// TIA Portal V19 export
FUNCTION "Prod_O_ACT_Pop_&_O_TODO_Push" : DInt   // FC63, LAD
TITLE = POP ORDINE IN LAVORO (ACT) SU ARRAY ORDINI DA FARE (TODO)
// stored: SetENOAutomatically false
   VAR_TEMP
      RETVAL : DInt;
   END_VAR
BEGIN

REGION Network 1 (SCL): SPOSTA ACT SU TODO

   //@@@@@@@@@@@@@@@@@@@@@@@@@@@@@@@@@@@@@@@@@@@@@@@@@@@@@@@@@@@@@@@@@@@@@@@@@@@@@@@@@@@
   //
   // PUSH
   // 
   //@@@@@@@@@@@@@@@@@@@@@@@@@@@@@@@@@@@@@@@@@@@@@@@@@@@@@@@@@@@@@@@@@@@@@@@@@@@@@@@@@@@


   #RETVAL :="PROD_item_Push_to_Top"(item := "Production".O_ACT , Evaluate_FULL := true, Buffer := "Production".O_TODO);


   IF #RETVAL < 0 THEN

       #"Prod_O_ACT_Pop_&_O_TODO_Push" := #RETVAL;

   END_IF;



   //@@@@@@@@@@@@@@@@@@@@@@@@@@@@@@@@@@@@@@@@@@@@@@@@@@@@@@@@@@@@@@@@@@@@@@@@@@@@@@@@@@@
   //
   // POP
   // 
   //@@@@@@@@@@@@@@@@@@@@@@@@@@@@@@@@@@@@@@@@@@@@@@@@@@@@@@@@@@@@@@@@@@@@@@@@@@@@@@@@@@@


   #RETVAL := "Prod_O_ACT_Pop"();


   // Uscita per errore OP
   // 
   IF #RETVAL < 0 THEN

       #"Prod_O_ACT_Pop_&_O_TODO_Push" := #RETVAL;

   END_IF;



   //@@@@@@@@@@@@@@@@@@@@@@@@@@@@@@@@@@@@@@@@@@@@@@@@@@@@@@@@@@@@@@@@@@@@@@@@@@@@@@@@@@@
   //
   // OK
   // 
   //@@@@@@@@@@@@@@@@@@@@@@@@@@@@@@@@@@@@@@@@@@@@@@@@@@@@@@@@@@@@@@@@@@@@@@@@@@@@@@@@@@@

   #"Prod_O_ACT_Pop_&_O_TODO_Push" := "PROD_FUN_RESULT_OK";
END_REGION
END_FUNCTION
